Universal Robots PolyScope program: Box_Demo.urp

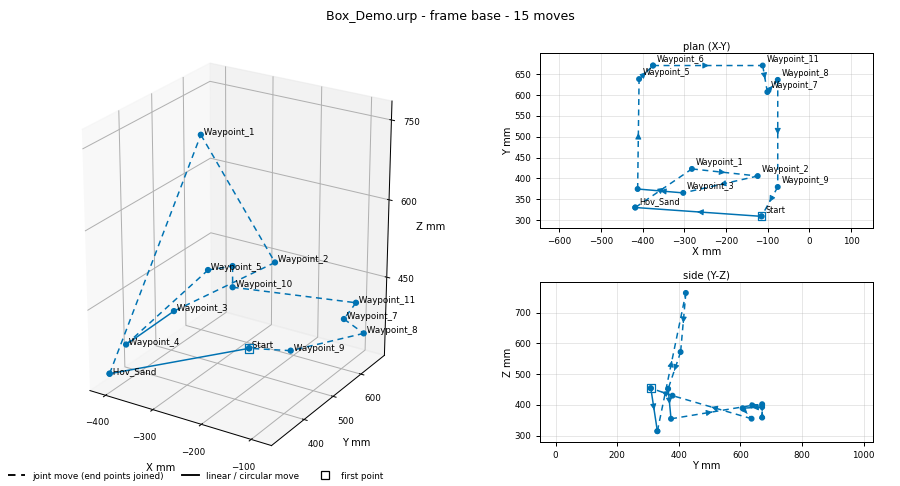
[picture p0: tool path of Box_Demo.urp in frame base, 15 of 15 moves have a stored position in this frame; points joined in program order, loops and branches not executed]
Program Box_Demo (installation=default directory=/programs/archive createdIn=5.11.5.1010327 lastSavedIn=5.11.5.1010327 robotSerialNumber=20215500677)
Calibrated DH parameters: a=[0.000204, -0.239222, -0.391845, -0.000001, 0.000022, 0]; d=[0.162722, -355.808559, 353.37206, 2.570385, 0.099741, 0.099629]; alpha=[1.571124, 0.000988, 0.008295, 1.568963, -1.570303, 0]; deltaTheta=[0, -0.973091, 7.204745, 0.05153, 0, 0]
Robot Program (runOnlyOnce=false)
  MoveL speed 250 mm/s, acceleration 1200 mm/s^2 (useActiveTCP=true) feature=Base
    Waypoint Start: TCP in base x=-114.851 y=309.141 z=454.167 mm, rx=-3.1183 ry=0.3817 rz=0 rad; joints [134.455, -65.585, -98.448, -105.996, 90.474, 58.151] deg; TCP offset x=0 y=0 z=105 mm, rx=0 ry=0 rz=0 rad
    Waypoint Hov_Sand: TCP in base x=-417.592 y=330.357 z=314.681 mm, rx=-3.1267 ry=0.3041 rz=0.0003 rad; joints [156.236, -93.888, -96.19, -79.939, 90.491, 77.317] deg
    URCap Zero FT Sensor (Robotiq_Copilot, Robotiq Inc.) dataModel(NodeInitializedKey=true, WaitForSteadyWrenchOptionKey=true)
    URCap Finishing Tool Control (Robotiq_Copilot, Robotiq Inc.) dataModel(ToolOutputNameKey=digital_out[4], HackTriggeringContributionIsDefinedMethodKey=true)
    Force Simple feature=Joint_6_name; selection=[0, 0, 1, 0, 0, 0]; wrench=[0, 0, 10, 0, 0, 0]; limitsForce=[0.15, 0.15, 0.15, 1.047198, 1.047198, 1.047198]; limitsMotion=[0.1, 0.1, 0.1, 0.349066, 0.349066, 0.349066]
      URCap Path Generator (Robotiq_Copilot, Robotiq Inc.) dataModel(pathOptionsTypeKey=TOOL_ON_ROBOT, coverageModeKey=PERIMETER_ONLY, PathTypeKey=FOUR_POINTS_VERTICAL, WaypointPoseKey2=[-0.41757674202011175, 0.6591609922755547, 0.30816835501828, -3.1266138859230534, 0.3040381995226014, 2.4995958662367575E-4], WaypointJointPositionsKey2=[2.307923930212736, -2.2813740978498203, -0.7922447768628365, -1.6390348210366525, 1.579702206231814, 0.9291134373511207], WaypointPoseKey1=[-0.4175788958663728, 0.33036542303365934, 0.3024547885572979, -3.1266923772008854, 0.3041148136239429, 3.199859133255452E-4], WaypointJointPositionsKey1=[2.7268086187595086, -1.6440882080001593, -1.7047043935521096, -1.3638269454445053, 1.5792601106647295, 1.3496651243599416], WaypointPoseKey3=[-0.062367863288705534, 0.33036121432411475, 0.30243995867730755, -3.126716087026817, 0.3040172129434159, 2.6437399106756415E-4], WaypointJointPositionsKey3=[2.168097809065898, -1.1282043766143426, -2.1177542442379256, -1.4666612935676575, 1.579235331304588, 0.7897625328574662], WaypointPoseKey4=[-0.06238273621350593, 0.6738181536675374, 0.3080769905516868, -3.1266307850380697, 0.3039862434956835, 3.375756405364136E-4], WaypointJointPositionsKey4=[1.8622899464339184, -1.9893917788467936, -1.2532328774484514, -1.4700298078215042, 1.5797898818581313, 0.4846028147601933], PerimeterSpeedKey=60, urcapVersion=1.22.1); state(isChildrenLocked=true)
        URCap Point (Robotiq_Copilot, Robotiq Inc.) dataModel(pose=[-0.4175788958663728, 0.33036542303365934, 0.3024547885572979, -3.1266923772008854, 0.3041148136239429, 3.199859133255452E-4], joint_positions=[2.7268086187595086, -1.6440882080001593, -1.7047043935521096, -1.3638269454445053, 1.5792601106647295, 1.3496651243599416])
        URCap Point (Robotiq_Copilot, Robotiq Inc.) dataModel(pose=[-0.41757674202011175, 0.6591609922755547, 0.30816835501828, -3.1266138859230534, 0.3040381995226014, 2.4995958662367575E-4], joint_positions=[2.307923930212736, -2.2813740978498203, -0.7922447768628365, -1.6390348210366525, 1.579702206231814, 0.9291134373511207])
        URCap Point (Robotiq_Copilot, Robotiq Inc.) dataModel(pose=[-0.062367863288705534, 0.33036121432411475, 0.30243995867730755, -3.126716087026817, 0.3040172129434159, 2.6437399106756415E-4], joint_positions=[2.168097809065898, -1.1282043766143426, -2.1177542442379256, -1.4666612935676575, 1.579235331304588, 0.7897625328574662])
        URCap Point (Robotiq_Copilot, Robotiq Inc.) dataModel(pose=[-0.06238273621350593, 0.6738181536675374, 0.3080769905516868, -3.1266307850380697, 0.3039862434956835, 3.375756405364136E-4], joint_positions=[1.8622899464339184, -1.9893917788467936, -1.2532328774484514, -1.4700298078215042, 1.5797898818581313, 0.4846028147601933])
    SuppressedNode
      URCap Force Control (Robotiq_Copilot, Robotiq Inc.) dataModel(NodeInitializedKey=true, force_x=0, force_y=0, force_mx=0, force_my=0, force_mz=0, limit_x_neg=-100, limit_y_neg=-100, limit_z_neg=-100, limit_x_pos=100, limit_y_pos=100, limit_z_pos=100, limit_mx_neg=-20, limit_my_neg=-20, limit_mz_neg=-20, limit_mx_pos=20, limit_my_pos=20, limit_mz_pos=20, ft_control_x=false, ft_control_y=false, ft_control_mx=false, ft_control_my=false, ft_control_mz=false, stiffness_x=100, stiffness_y=100, stiffness_z_position=100, stiffness_mx=100, stiffness_my=100, stiffness_mz=100, adaptive_stiffness=true, is_force_control_about_actual_position=true, HackTriggeringContributionIsDefinedMethodKey=true, ft_control_z=true, force_z=15, TranslatableFeatureKey=1)
        URCap Path Generator (Robotiq_Copilot, Robotiq Inc.) dataModel(pathOptionsTypeKey=TOOL_ON_ROBOT, coverageModeKey=PERIMETER_ONLY, PathTypeKey=FOUR_POINTS_VERTICAL, WaypointPoseKey2=[-0.41757674202011175, 0.6591609922755547, 0.30816835501828, -3.1266138859230534, 0.3040381995226014, 2.4995958662367575E-4], WaypointJointPositionsKey2=[2.307923930212736, -2.2813740978498203, -0.7922447768628365, -1.6390348210366525, 1.579702206231814, 0.9291134373511207], WaypointPoseKey1=[-0.4175788958663728, 0.33036542303365934, 0.3024547885572979, -3.1266923772008854, 0.3041148136239429, 3.199859133255452E-4], WaypointJointPositionsKey1=[2.7268086187595086, -1.6440882080001593, -1.7047043935521096, -1.3638269454445053, 1.5792601106647295, 1.3496651243599416], WaypointPoseKey3=[-0.062367863288705534, 0.33036121432411475, 0.30243995867730755, -3.126716087026817, 0.3040172129434159, 2.6437399106756415E-4], WaypointJointPositionsKey3=[2.168097809065898, -1.1282043766143426, -2.1177542442379256, -1.4666612935676575, 1.579235331304588, 0.7897625328574662], WaypointPoseKey4=[-0.06238273621350593, 0.6738181536675374, 0.3080769905516868, -3.1266307850380697, 0.3039862434956835, 3.375756405364136E-4], WaypointJointPositionsKey4=[1.8622899464339184, -1.9893917788467936, -1.2532328774484514, -1.4700298078215042, 1.5797898818581313, 0.4846028147601933], PerimeterSpeedKey=60, urcapVersion=1.22.1); state(isChildrenLocked=true)
          URCap Point (Robotiq_Copilot, Robotiq Inc.) dataModel(pose=[-0.4175788958663728, 0.33036542303365934, 0.3024547885572979, -3.1266923772008854, 0.3041148136239429, 3.199859133255452E-4], joint_positions=[2.7268086187595086, -1.6440882080001593, -1.7047043935521096, -1.3638269454445053, 1.5792601106647295, 1.3496651243599416])
          URCap Point (Robotiq_Copilot, Robotiq Inc.) dataModel(pose=[-0.41757674202011175, 0.6591609922755547, 0.30816835501828, -3.1266138859230534, 0.3040381995226014, 2.4995958662367575E-4], joint_positions=[2.307923930212736, -2.2813740978498203, -0.7922447768628365, -1.6390348210366525, 1.579702206231814, 0.9291134373511207])
          URCap Point (Robotiq_Copilot, Robotiq Inc.) dataModel(pose=[-0.062367863288705534, 0.33036121432411475, 0.30243995867730755, -3.126716087026817, 0.3040172129434159, 2.6437399106756415E-4], joint_positions=[2.168097809065898, -1.1282043766143426, -2.1177542442379256, -1.4666612935676575, 1.579235331304588, 0.7897625328574662])
          URCap Point (Robotiq_Copilot, Robotiq Inc.) dataModel(pose=[-0.06238273621350593, 0.6738181536675374, 0.3080769905516868, -3.1266307850380697, 0.3039862434956835, 3.375756405364136E-4], joint_positions=[1.8622899464339184, -1.9893917788467936, -1.2532328774484514, -1.4700298078215042, 1.5797898818581313, 0.4846028147601933])
    URCap Finishing Tool Control (Robotiq_Copilot, Robotiq Inc.) dataModel(FinishingToolStateKey=false, ToolOutputNameKey=digital_out[4], HackTriggeringContributionIsDefinedMethodKey=true)
    Waypoint Hov_Sand: TCP in base x=-417.592 y=330.357 z=314.681 mm, rx=-3.1267 ry=0.3041 rz=0.0003 rad; joints [156.236, -93.888, -96.19, -79.939, 90.491, 77.317] deg
  MoveJ speed 60 deg/s, acceleration 80 deg/s^2 (useActiveTCP=true) feature=Base
    Waypoint Waypoint_1: motionParameters(blendRadius=0.005); TCP in base x=-281.745 y=422.892 z=763.813 mm, rx=-0.7767 ry=0.9376 rz=1.9667 rad; joints [156.194, -90.928, -89.502, 47.28, 46.611, 77.071] deg
    Waypoint Waypoint_2: motionParameters(blendRadius=0.005); TCP in base x=-123.93 y=405.832 z=571.918 mm, rx=-1.2629 ry=-2.1158 rz=-1.5876 rad; joints [156.213, -87.111, -81.05, 87.167, -24.26, 122.055] deg
    Waypoint Waypoint_3: TCP in base x=-302.523 y=365.386 z=452.292 mm, rx=1.595 ry=-2.4399 rz=-0.5648 rad; joints [145.707, -101.408, -63.94, 99.395, -91.274, -10.275] deg
  MoveL speed 250 mm/s, acceleration 1200 mm/s^2 (useActiveTCP=true) feature=Base
    Waypoint Waypoint_4: TCP in base x=-411.831 y=374.715 z=354.928 mm, rx=1.0225 ry=-1.3174 rz=-1.0225 rad; joints [137.318, -94.802, -104.977, 200.349, -132.524, 15.176] deg
  URCap Finishing Tool Control (Robotiq_Copilot, Robotiq Inc.) dataModel(FinishingToolStateKey=true, ToolOutputNameKey=digital_out[4], HackTriggeringContributionIsDefinedMethodKey=true)
  Force Simple feature=Joint_6_name; selection=[0, 0, 1, 0, 0, 0]; wrench=[0, 0, 7, 0, 0, 0]; limitsForce=[0.15, 0.15, 0.15, 1.047198, 1.047198, 1.047198]; limitsMotion=[0.1, 0.1, 0.1, 0.349066, 0.349066, 0.349066]
    URCap Multipoint Path (Robotiq_Copilot, Robotiq Inc.) dataModel(NodeInitializedKey=true, pathOptionsTypeKey=TOOL_ON_ROBOT, SPEED_VALUE=60, waypointIndexKey=2, HackTriggeringContributionIsDefinedMethodKey=true, urcapVersion=1.22.1)
      URCap Waypoint (Robotiq_Copilot, Robotiq Inc.) dataModel(pose=[-0.4118426791032656, 0.37470264736820286, 0.35494420079657746, 1.0224642144428697, -1.3173851925939044, -1.0224911221945254], jointPositions=[2.3966512700782423, -1.6546012378153856, -1.832199571966929, 3.4967433647850226, -2.312975468082811, 0.2648702859925189], waypointType=CURVE, waypointIndex=0, initialized=true, NodeIndexKey=1, RenamedTitleKey=UnrenamedTitle, urcapVersion=1.22.1)
      URCap Waypoint (Robotiq_Copilot, Robotiq Inc.) dataModel(NodeIndexKey=2, RenamedTitleKey=UnrenamedTitle, pose=[-0.4118456043740054, 0.6384093063872077, 0.3549149040540559, 1.0225066070735933, -1.3173709096907638, -1.0224574119347611], jointPositions=[2.086801139600663, -2.2439716834894803, -1.003929292486963, 3.2677811105189463, -2.624130895568669, 0.27333331071319156], waypointType=LINE, waypointIndex=0, initialized=true, urcapVersion=1.22.1)
  SuppressedNode
    URCap Force Control (Robotiq_Copilot, Robotiq Inc.) dataModel(NodeInitializedKey=true, force_x=0, force_y=0, force_mx=0, force_my=0, force_mz=0, limit_x_neg=-100, limit_y_neg=-100, limit_z_neg=-100, limit_x_pos=100, limit_y_pos=100, limit_z_pos=100, limit_mx_neg=-20, limit_my_neg=-20, limit_mz_neg=-20, limit_mx_pos=20, limit_my_pos=20, limit_mz_pos=20, ft_control_x=false, ft_control_y=false, ft_control_mx=false, ft_control_my=false, ft_control_mz=false, stiffness_x=100, stiffness_y=100, stiffness_z_position=100, stiffness_mx=100, stiffness_my=100, stiffness_mz=100, adaptive_stiffness=true, is_force_control_about_actual_position=true, HackTriggeringContributionIsDefinedMethodKey=true, ft_control_z=true, force_z=15, TranslatableFeatureKey=1)
      URCap Multipoint Path (Robotiq_Copilot, Robotiq Inc.) dataModel(NodeInitializedKey=true, pathOptionsTypeKey=TOOL_ON_ROBOT, HackTriggeringContributionIsDefinedMethodKey=true, SPEED_VALUE=60, waypointIndexKey=2, urcapVersion=1.22.1)
        URCap Waypoint (Robotiq_Copilot, Robotiq Inc.) dataModel(pose=[-0.4118426791032656, 0.37470264736820286, 0.35494420079657746, 1.0224642144428697, -1.3173851925939044, -1.0224911221945254], jointPositions=[2.3966512700782423, -1.6546012378153856, -1.832199571966929, 3.4967433647850226, -2.312975468082811, 0.2648702859925189], waypointType=CURVE, waypointIndex=0, initialized=true, NodeIndexKey=1, RenamedTitleKey=UnrenamedTitle, urcapVersion=1.22.1)
        URCap Waypoint (Robotiq_Copilot, Robotiq Inc.) dataModel(NodeIndexKey=2, RenamedTitleKey=UnrenamedTitle, pose=[-0.4118456043740054, 0.6384093063872077, 0.3549149040540559, 1.0225066070735933, -1.3173709096907638, -1.0224574119347611], jointPositions=[2.086801139600663, -2.2439716834894803, -1.003929292486963, 3.2677811105189463, -2.624130895568669, 0.27333331071319156], waypointType=LINE, waypointIndex=0, initialized=true, urcapVersion=1.22.1)
  URCap Finishing Tool Control (Robotiq_Copilot, Robotiq Inc.) dataModel(FinishingToolStateKey=false, ToolOutputNameKey=digital_out[4], HackTriggeringContributionIsDefinedMethodKey=true)
  MoveJ speed 60 deg/s, acceleration 80 deg/s^2 (useActiveTCP=true) feature=Base
    Waypoint Waypoint_5: motionParameters(blendRadius=0.005); TCP in base x=-408.416 y=638.33 z=398.706 mm, rx=1.0225 ry=-1.3173 rz=-1.0224 rad; joints [119.308, -128.008, -52.058, 181.228, -150.667, 15.684] deg
    Waypoint Waypoint_6: TCP in base x=-374.971 y=670.758 z=402.321 mm, rx=-0.0001 ry=2.2215 rz=2.2213 rad; joints [141.844, -117.071, -68.834, 185.163, -38.093, 0.956] deg
    Waypoint Waypoint_10: TCP in base x=-374.941 y=670.767 z=358.855 mm, rx=0.0002 ry=2.2213 rz=2.2215 rad; joints [141.843, -118.003, -73.859, 191.149, -38.038, 0.938] deg
    URCap Finishing Tool Control (Robotiq_Copilot, Robotiq Inc.) dataModel(ToolOutputNameKey=digital_out[4], HackTriggeringContributionIsDefinedMethodKey=true, FinishingToolStateKey=true)
  SuppressedNode
    URCap Force Control (Robotiq_Copilot, Robotiq Inc.) dataModel(NodeInitializedKey=true, force_x=0, force_y=0, force_mx=0, force_my=0, force_mz=0, limit_x_neg=-100, limit_y_neg=-100, limit_z_neg=-100, limit_x_pos=100, limit_y_pos=100, limit_z_pos=100, limit_mx_neg=-20, limit_my_neg=-20, limit_mz_neg=-20, limit_mx_pos=20, limit_my_pos=20, limit_mz_pos=20, ft_control_x=false, ft_control_y=false, ft_control_mx=false, ft_control_my=false, ft_control_mz=false, stiffness_x=100, stiffness_y=100, stiffness_z_position=100, stiffness_mx=100, stiffness_my=100, stiffness_mz=100, adaptive_stiffness=true, is_force_control_about_actual_position=true, HackTriggeringContributionIsDefinedMethodKey=true, ft_control_z=true, force_z=15, TranslatableFeatureKey=1)
      URCap Multipoint Path (Robotiq_Copilot, Robotiq Inc.) dataModel(NodeInitializedKey=true, pathOptionsTypeKey=TOOL_ON_ROBOT, HackTriggeringContributionIsDefinedMethodKey=true, SPEED_VALUE=60, waypointIndexKey=2, urcapVersion=1.22.1)
        URCap Waypoint (Robotiq_Copilot, Robotiq Inc.) dataModel(NodeIndexKey=1, RenamedTitleKey=UnrenamedTitle, pose=[-0.374931293716131, 0.6707707844931435, 0.35826453275846937, -8.685668482526667E-6, 2.2213708525814324, 2.2213969867533074], jointPositions=[2.4756537233251112, -2.059888285471577, -1.290110463452411, 3.337379944306388, -0.663960923454356, 0.016377029988271667], waypointType=CURVE, waypointIndex=0, initialized=true, urcapVersion=1.22.1)
        URCap Waypoint (Robotiq_Copilot, Robotiq Inc.) dataModel(NodeIndexKey=2, RenamedTitleKey=UnrenamedTitle, pose=[-0.11198786447953216, 0.6707641984985253, 0.3582390946310843, -4.681852097414058E-5, 2.221413533566073, 2.221425284772222], jointPositions=[2.0920012458238606, -1.7770066793724482, -1.680655228331096, 3.4523736784688652, -1.0470068768474299, 0.011406973830797362], waypointType=LINE, waypointIndex=0, initialized=true, urcapVersion=1.22.1)
  Force Simple feature=Joint_6_name; selection=[0, 0, 1, 0, 0, 0]; wrench=[0, 0, 7, 0, 0, 0]; limitsForce=[0.15, 0.15, 0.15, 1.047198, 1.047198, 1.047198]; limitsMotion=[0.1, 0.1, 0.1, 0.349066, 0.349066, 0.349066]
    URCap Multipoint Path (Robotiq_Copilot, Robotiq Inc.) dataModel(NodeInitializedKey=true, pathOptionsTypeKey=TOOL_ON_ROBOT, SPEED_VALUE=60, waypointIndexKey=2, HackTriggeringContributionIsDefinedMethodKey=true, urcapVersion=1.22.1)
      URCap Waypoint (Robotiq_Copilot, Robotiq Inc.) dataModel(NodeIndexKey=1, RenamedTitleKey=UnrenamedTitle, pose=[-0.37493230762041424, 0.6707901929328213, 0.3588601739332959, -2.641988741817746E-4, -2.2212357412106885, -2.221558615803627], jointPositions=[2.4755976999660905, -2.059559411764874, -1.289103005258876, 3.336195783900461, -0.6639509409143365, 0.01637744255208911], waypointType=CURVE, waypointIndex=0, initialized=true, urcapVersion=1.22.1)
      URCap Waypoint (Robotiq_Copilot, Robotiq Inc.) dataModel(NodeIndexKey=2, RenamedTitleKey=UnrenamedTitle, pose=[-0.11244759839429963, 0.670776367352553, 0.35888767524115806, -1.9202562664255975E-4, -2.2211821066375315, -2.221607170577835], jointPositions=[2.092782472646748, -1.7768432265496088, -1.6793063277095275, 3.450958635604234, -1.0461609183412115, 0.011480200840463084], waypointType=LINE, waypointIndex=0, initialized=true, urcapVersion=1.22.1)
  URCap Finishing Tool Control (Robotiq_Copilot, Robotiq Inc.) dataModel(FinishingToolStateKey=false, ToolOutputNameKey=digital_out[4], HackTriggeringContributionIsDefinedMethodKey=true)
  MoveJ speed 60 deg/s, acceleration 80 deg/s^2 (useActiveTCP=true) feature=Base
    Waypoint Waypoint_11: TCP in base x=-111.997 y=670.77 z=393.054 mm, rx=-0.0002 ry=2.2214 rz=2.2214 rad; joints [119.862, -100.564, -92.541, 192.794, -60.033, 0.665] deg
    Waypoint Waypoint_7: motionParameters(blendRadius=0.005); TCP in base x=-100.897 y=607.259 z=389.405 mm, rx=1.1249 ry=1.4463 rz=1.0148 rad; joints [128.385, -124.371, -55.448, 194.753, 37.255, -24.474] deg
    Waypoint Waypoint_8: TCP in base x=-75.923 y=636.359 z=355.317 mm, rx=0.9574 ry=1.35 rz=0.9574 rad; joints [124.964, -132.77, -50.287, 183.889, 35.026, -20.347] deg
    URCap Finishing Tool Control (Robotiq_Copilot, Robotiq Inc.) dataModel(ToolOutputNameKey=digital_out[4], HackTriggeringContributionIsDefinedMethodKey=true, FinishingToolStateKey=true)
  SuppressedNode
    URCap Force Control (Robotiq_Copilot, Robotiq Inc.) dataModel(NodeInitializedKey=true, force_x=0, force_y=0, force_mx=0, force_my=0, force_mz=0, limit_x_neg=-100, limit_y_neg=-100, limit_z_neg=-100, limit_x_pos=100, limit_y_pos=100, limit_z_pos=100, limit_mx_neg=-20, limit_my_neg=-20, limit_mz_neg=-20, limit_mx_pos=20, limit_my_pos=20, limit_mz_pos=20, ft_control_x=false, ft_control_y=false, ft_control_mx=false, ft_control_my=false, ft_control_mz=false, stiffness_x=100, stiffness_y=100, stiffness_z_position=100, stiffness_mx=100, stiffness_my=100, stiffness_mz=100, adaptive_stiffness=true, is_force_control_about_actual_position=true, HackTriggeringContributionIsDefinedMethodKey=true, ft_control_z=true, force_z=15, TranslatableFeatureKey=1)
      URCap Multipoint Path (Robotiq_Copilot, Robotiq Inc.) dataModel(NodeInitializedKey=true, pathOptionsTypeKey=TOOL_ON_ROBOT, HackTriggeringContributionIsDefinedMethodKey=true, SPEED_VALUE=60, waypointIndexKey=2, urcapVersion=1.22.1)
        URCap Waypoint (Robotiq_Copilot, Robotiq Inc.) dataModel(pose=[-0.07592416617044802, 0.6363465379672868, 0.3553099409959876, 0.9574480501797192, 1.350020624397844, 0.9573465971042064], jointPositions=[2.1810557715665766, -2.317277683250932, -0.8777256208774933, 3.2094613813733144, 0.6113304911626471, -0.35513429454046275], waypointType=CURVE, waypointIndex=0, initialized=true, NodeIndexKey=1, RenamedTitleKey=UnrenamedTitle, urcapVersion=1.22.1)
        URCap Waypoint (Robotiq_Copilot, Robotiq Inc.) dataModel(NodeIndexKey=2, RenamedTitleKey=UnrenamedTitle, pose=[-0.07591897906080214, 0.3795684818444538, 0.35531699361886754, 0.9574351132459505, 1.3499940656618366, 0.9573077961733287], jointPositions=[2.497374662501389, -1.7590779390841336, -1.7104681325034772, 3.476501376841887, 0.929283824121991, -0.34939838032203596], waypointType=LINE, waypointIndex=0, initialized=true, urcapVersion=1.22.1)
  Force Simple feature=Joint_6_name; selection=[0, 0, 1, 0, 0, 0]; wrench=[0, 0, 7, 0, 0, 0]; limitsForce=[0.15, 0.15, 0.15, 1.047198, 1.047198, 1.047198]; limitsMotion=[0.1, 0.1, 0.1, 0.349066, 0.349066, 0.349066]
    URCap Multipoint Path (Robotiq_Copilot, Robotiq Inc.) dataModel(NodeInitializedKey=true, pathOptionsTypeKey=TOOL_ON_ROBOT, SPEED_VALUE=60, waypointIndexKey=2, HackTriggeringContributionIsDefinedMethodKey=true, urcapVersion=1.22.1)
      URCap Waypoint (Robotiq_Copilot, Robotiq Inc.) dataModel(pose=[-0.07592416617044802, 0.6363465379672868, 0.3553099409959876, 0.9574480501797192, 1.350020624397844, 0.9573465971042064], jointPositions=[2.1810557715665766, -2.317277683250932, -0.8777256208774933, 3.2094613813733144, 0.6113304911626471, -0.35513429454046275], waypointType=CURVE, waypointIndex=0, initialized=true, NodeIndexKey=1, RenamedTitleKey=UnrenamedTitle, urcapVersion=1.22.1)
      URCap Waypoint (Robotiq_Copilot, Robotiq Inc.) dataModel(NodeIndexKey=2, RenamedTitleKey=UnrenamedTitle, pose=[-0.07591897906080214, 0.3795684818444538, 0.35531699361886754, 0.9574351132459505, 1.3499940656618366, 0.9573077961733287], jointPositions=[2.497374662501389, -1.7590779390841336, -1.7104681325034772, 3.476501376841887, 0.929283824121991, -0.34939838032203596], waypointType=LINE, waypointIndex=0, initialized=true, urcapVersion=1.22.1)
  URCap Finishing Tool Control (Robotiq_Copilot, Robotiq Inc.) dataModel(FinishingToolStateKey=false, ToolOutputNameKey=digital_out[4], HackTriggeringContributionIsDefinedMethodKey=true)
  MoveJ speed 60 deg/s, acceleration 80 deg/s^2 (useActiveTCP=true) feature=Base
    Waypoint Waypoint_9: motionParameters(blendRadius=0.01); TCP in base x=-75.948 y=379.576 z=430.163 mm, rx=0.9574 ry=1.35 rz=0.9573 rad; joints [143.093, -98.472, -89.504, 188.395, 53.162, -20.051] deg
    Waypoint Start: TCP in base x=-114.851 y=309.141 z=454.167 mm, rx=-3.1183 ry=0.3817 rz=0 rad; joints [134.455, -65.585, -98.448, -105.996, 90.474, 58.151] deg
